// Mitsubishi GX Works2 project: PRJ_TEST   PLC: Q03UDV

PROGRAM MAIN
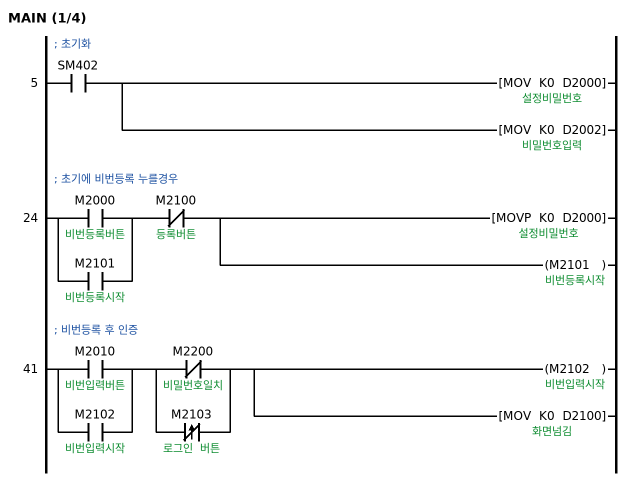
; 초기화
5     LD      SM402
      MOV     K0 D2000  ; 설정비밀번호
      MOV     K0 D2002  ; 비밀번호입력
; 초기에 비번등록 누를경우
24    LD      M2000  ; 비번등록버튼
      OR      M2101  ; 비번등록시작
      ANI     M2100  ; 등록버튼
      MOVP    K0 D2000
      OUT     M2101  ; 비번등록시작
; 비번등록 후 인증
41    LD      M2010  ; 비번입력버튼
      OR      M2102  ; 비번입력시작
      LDI     M2200  ; 비밀번호일치
      ORPI    M2103  ; 로그인  버튼
      ANB
      OUT     M2102  ; 비번입력시작
      MOV     K0 D2100  ; 화면넘김
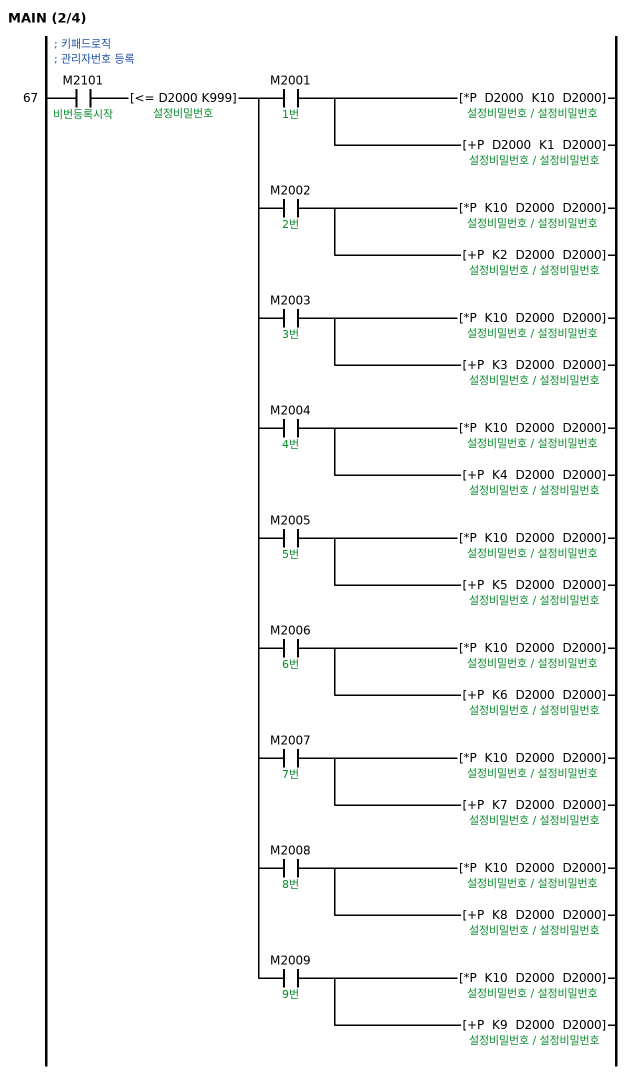
; 키패드로직
; 관리자번호 등록
67    LD      M2101  ; 비번등록시작
      AND<=   D2000 K999  ; 설정비밀번호
      MPS
      AND     M2001  ; 1번
      *P      D2000 K10 D2000
      +P      D2000 K1 D2000
      MRD
      AND     M2002  ; 2번
      *P      K10 D2000 D2000
      +P      K2 D2000 D2000
      MRD
      AND     M2003  ; 3번
      *P      K10 D2000 D2000
      +P      K3 D2000 D2000
      MRD
      AND     M2004  ; 4번
      *P      K10 D2000 D2000
      +P      K4 D2000 D2000
      MRD
      AND     M2005  ; 5번
      *P      K10 D2000 D2000
      +P      K5 D2000 D2000
      MRD
      AND     M2006  ; 6번
      *P      K10 D2000 D2000
      +P      K6 D2000 D2000
      MRD
      AND     M2007  ; 7번
      *P      K10 D2000 D2000
      +P      K7 D2000 D2000
      MRD
      AND     M2008  ; 8번
      *P      K10 D2000 D2000
      +P      K8 D2000 D2000
      MPP
      AND     M2009  ; 9번
      *P      K10 D2000 D2000
      +P      K9 D2000 D2000
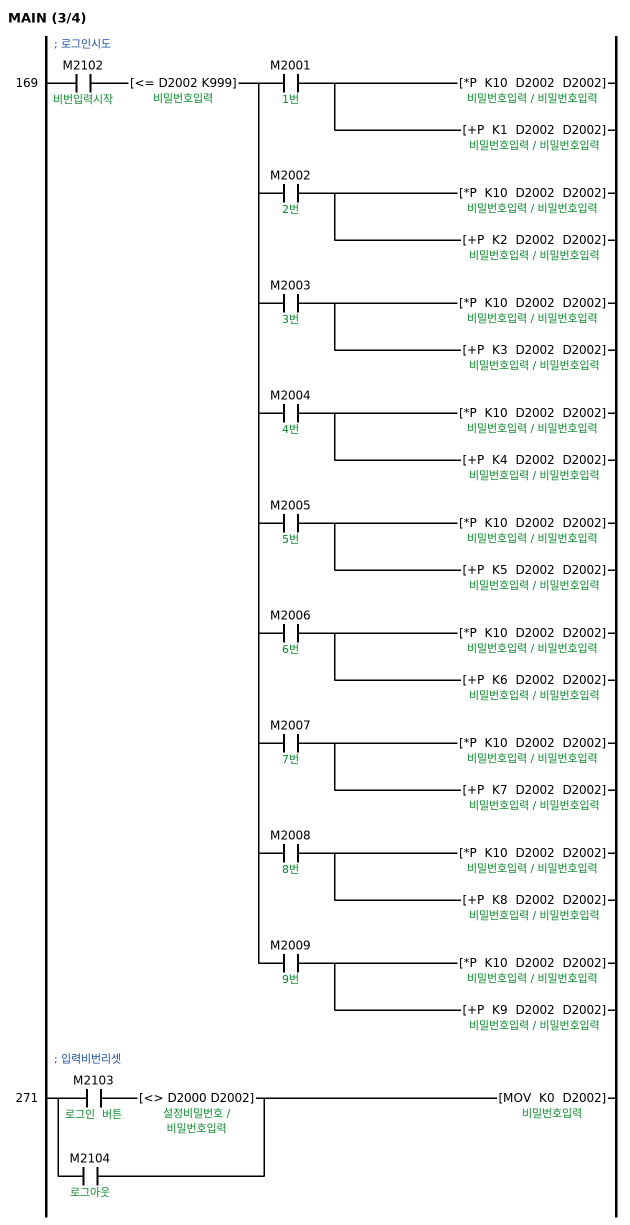
; 로그인시도
169   LD      M2102  ; 비번입력시작
      AND<=   D2002 K999  ; 비밀번호입력
      MPS
      AND     M2001  ; 1번
      *P      K10 D2002 D2002
      +P      K1 D2002 D2002
      MRD
      AND     M2002  ; 2번
      *P      K10 D2002 D2002
      +P      K2 D2002 D2002
      MRD
      AND     M2003  ; 3번
      *P      K10 D2002 D2002
      +P      K3 D2002 D2002
      MRD
      AND     M2004  ; 4번
      *P      K10 D2002 D2002
      +P      K4 D2002 D2002
      MRD
      AND     M2005  ; 5번
      *P      K10 D2002 D2002
      +P      K5 D2002 D2002
      MRD
      AND     M2006  ; 6번
      *P      K10 D2002 D2002
      +P      K6 D2002 D2002
      MRD
      AND     M2007  ; 7번
      *P      K10 D2002 D2002
      +P      K7 D2002 D2002
      MRD
      AND     M2008  ; 8번
      *P      K10 D2002 D2002
      +P      K8 D2002 D2002
      MPP
      AND     M2009  ; 9번
      *P      K10 D2002 D2002
      +P      K9 D2002 D2002
; 입력비번리셋
271   LD      M2103  ; 로그인  버튼
      AND<>   D2000 D2002  ; 설정비밀번호 / 비밀번호입력
      OR      M2104  ; 로그아웃
      MOV     K0 D2002
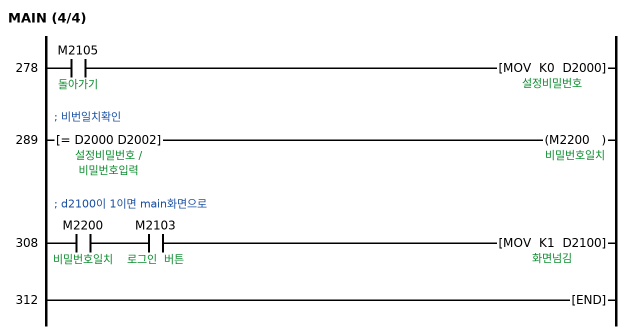
278   LD      M2105  ; 돌아가기
      MOV     K0 D2000
; 비번일치확인
289   LD=     D2000 D2002  ; 설정비밀번호 / 비밀번호입력
      OUT     M2200  ; 비밀번호일치
; d2100이 1이면 main화면으로
308   LD      M2200  ; 비밀번호일치
      AND     M2103  ; 로그인  버튼
      MOV     K1 D2100
312   END
END_PROGRAM

// device comments not shown above
D0  ; 설정비밀번호
D1  ; 입력비밀번호
D2  ; 비밀번호입력
D100  ; 화면넘김
M0  ; 비번등록버튼
M10  ; 비번입력버튼
M100  ; 등록버튼
M101  ; 비번등록시작
M102  ; 비번입력시작
M103  ; 승인버튼
M104  ; 로그아웃
M105  ; 등록하지않고 돌아가기
M200  ; 비밀번호 일치
M201  ; 다음페이지
